// SIMATIC S7-200 project (STEP 7-Micro/WIN), CPU 222 REL 01.22

SYMBOL_TABLE USR1
手动上升I            I0.0     // 用做手动上升，有故障时做故障复位用，常开
手动下降I            I0.1     // 用做手动下降，有故障时做故障复位用，常开
上限位I             I0.2     // 常闭
下限位I             I0.3     // 常闭
启动I              I0.4     // 常开
超时输入I            I0.5     // 来自转子短接接触器，常闭
超温输入I            I0.6     // 常开
上升输出Q            Q0.0     // 上升接触器
下降输出Q            Q0.1     // 下降接触器
允许起动Q            Q0.2     // 给高压柜的允许起动信号
超时跳闸Q            Q0.3     // 包括液体柜电极下降超时及短接接触器超时
转子短接Q            Q0.4
超温报警Q            Q0.5
上升中继M            M1.0     // 调用手动子程序过度用
下降中继M            M1.1     // 调用手动子程序过度用
起动中继M            M1.2     // 调用自动子程序过度用
定时搅拌M            M1.3     // 防止粉沉淀
END_SYMBOL_TABLE

ORGANIZATION_BLOCK 主:OB1
TITLE= 
// 程序注释
// 按 F1 获得帮助及举例程序
//  
BEGIN
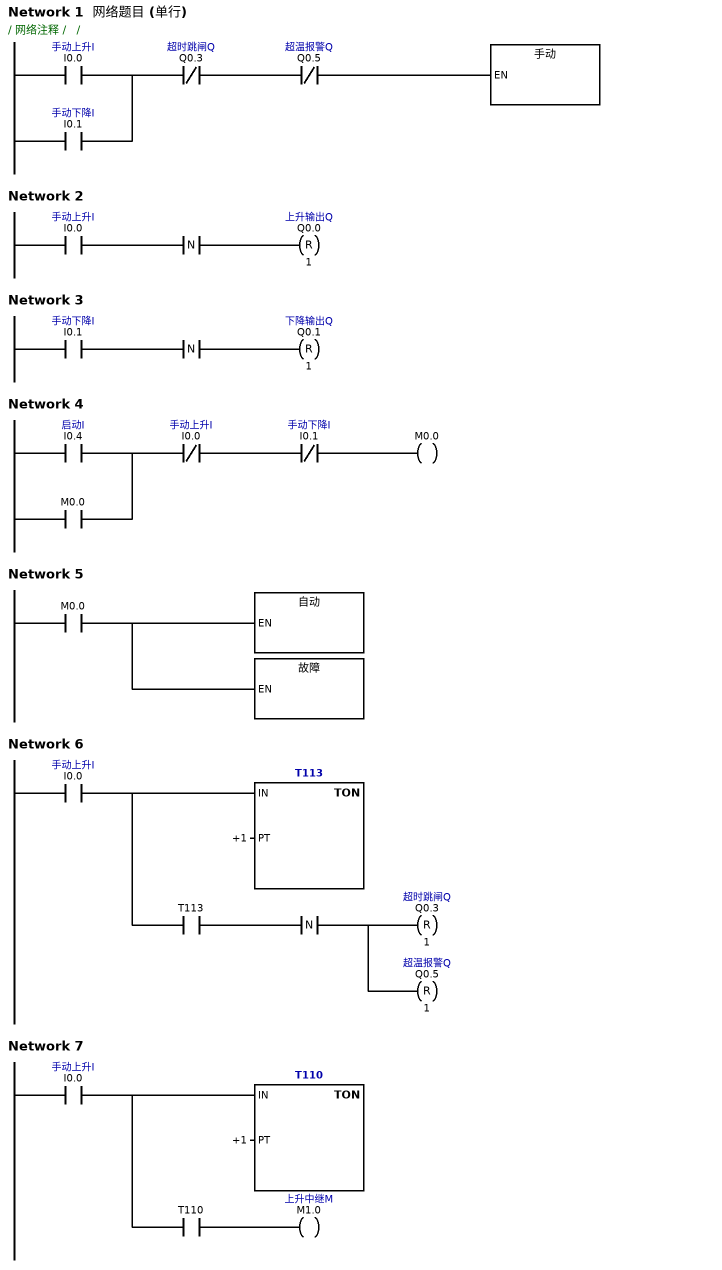
Network 1 // 网络题目 (单行)
//  
// 网络注释
//  
// 
// (network saved uncompiled; LAD cells follow)
// row 0: c0 -| |- 手动上升I:I0.0 v  c1 -|/|- 超时跳闸Q:Q0.3  c2 -|/|- 超温报警Q:Q0.5  c3 --  c4 [手动 EN:=power@row0]
// row 1: c0 -| |- 手动下降I:I0.1 ^
Network 2
// (network saved uncompiled; LAD cells follow)
// row 0: c0 -| |- 手动上升I:I0.0  c1 -|N|-  c2 -(R) 上升输出Q:Q0.0, 1
Network 3
// (network saved uncompiled; LAD cells follow)
// row 0: c0 -| |- 手动下降I:I0.1  c1 -|N|-  c2 -(R) 下降输出Q:Q0.1, 1
Network 4
// (network saved uncompiled; LAD cells follow)
// row 0: c0 -| |- 启动I:I0.4 v  c1 -|/|- 手动上升I:I0.0  c2 -|/|- 手动下降I:I0.1  c3 -( ) M0.0
// row 1: c0 -| |- M0.0 ^
Network 5
// (network saved uncompiled; LAD cells follow)
// row 0: c0 -| |- M0.0 v  c1 --  c2 [自动 EN:=power@row0]
// row 1: c0 ^  c1 --  c2 [故障 EN:=power@row1]
Network 6
// (network saved uncompiled; LAD cells follow)
// row 0: c0 -| |- 手动上升I:I0.0 v  c1 --  c2 [TON T113 IN:=power@row0, PT:=+1]
// row 1: c0 ^v  c2 [box]
// row 2: c0 ^  c1 -| |- T113  c2 -|N|-  v  c3 -(R) 超时跳闸Q:Q0.3, 1
// row 3: c2 ^  c3 -(R) 超温报警Q:Q0.5, 1
Network 7
// (network saved uncompiled; LAD cells follow)
// row 0: c0 -| |- 手动上升I:I0.0 v  c1 --  c2 [TON T110 IN:=power@row0, PT:=+1]
// row 1: c0 ^v  c2 [box]
// row 2: c0 ^  c1 -| |- T110  c2 -( ) 上升中继M:M1.0
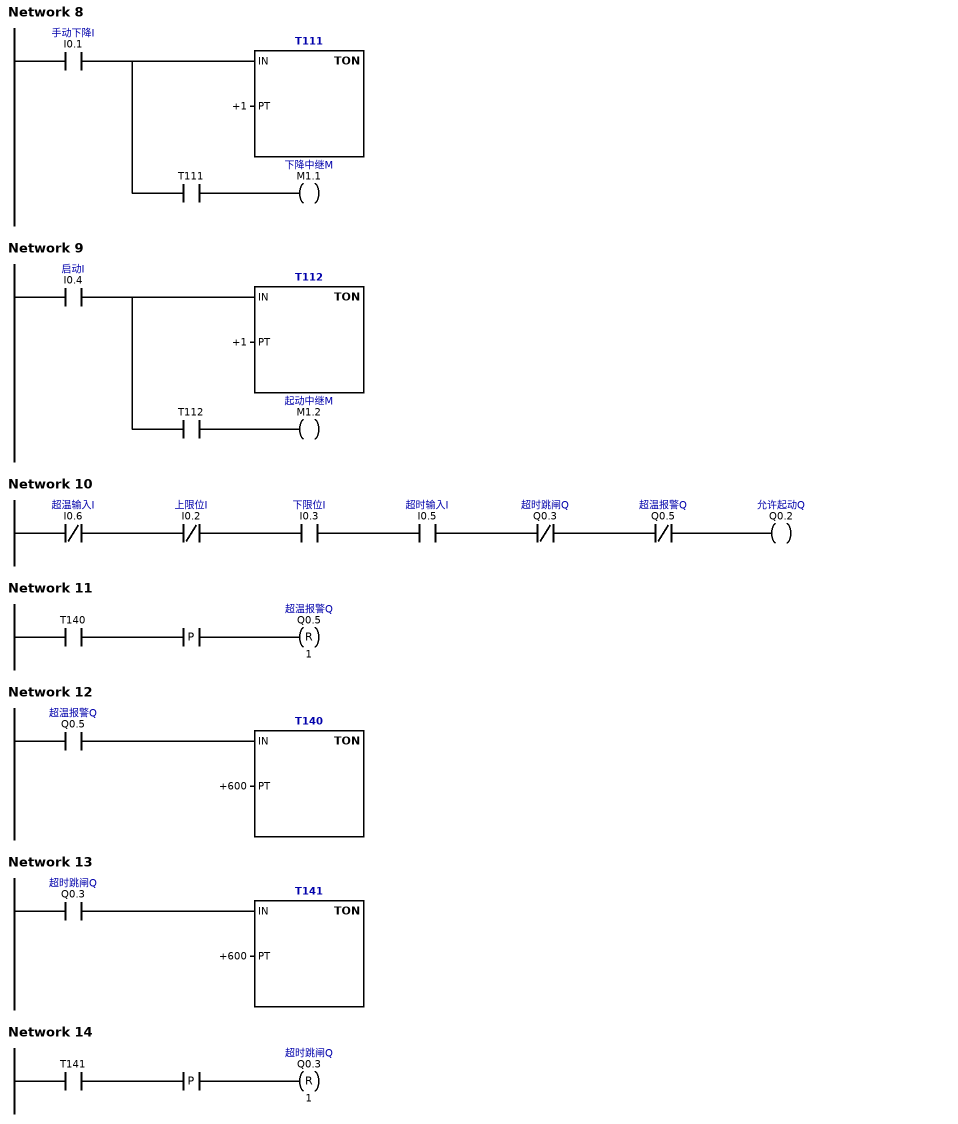
Network 8
// (network saved uncompiled; LAD cells follow)
// row 0: c0 -| |- 手动下降I:I0.1 v  c1 --  c2 [TON T111 IN:=power@row0, PT:=+1]
// row 1: c0 ^v  c2 [box]
// row 2: c0 ^  c1 -| |- T111  c2 -( ) 下降中继M:M1.1
Network 9
// (network saved uncompiled; LAD cells follow)
// row 0: c0 -| |- 启动I:I0.4 v  c1 --  c2 [TON T112 IN:=power@row0, PT:=+1]
// row 1: c0 ^v  c2 [box]
// row 2: c0 ^  c1 -| |- T112  c2 -( ) 起动中继M:M1.2
Network 10
// (network saved uncompiled; LAD cells follow)
// row 0: c0 -|/|- 超温输入I:I0.6  c1 -|/|- 上限位I:I0.2  c2 -| |- 下限位I:I0.3  c3 -| |- 超时输入I:I0.5  c4 -|/|- 超时跳闸Q:Q0.3  c5 -|/|- 超温报警Q:Q0.5  c6 -( ) 允许起动Q:Q0.2
Network 11
// (network saved uncompiled; LAD cells follow)
// row 0: c0 -| |- T140  c1 -|P|-  c2 -(R) 超温报警Q:Q0.5, 1
Network 12
// (network saved uncompiled; LAD cells follow)
// row 0: c0 -| |- 超温报警Q:Q0.5  c1 --  c2 [TON T140 IN:=power@row0, PT:=+600]
// row 1: c2 [box]
Network 13
// (network saved uncompiled; LAD cells follow)
// row 0: c0 -| |- 超时跳闸Q:Q0.3  c1 --  c2 [TON T141 IN:=power@row0, PT:=+600]
// row 1: c2 [box]
Network 14
// (network saved uncompiled; LAD cells follow)
// row 0: c0 -| |- T141  c1 -|P|-  c2 -(R) 超时跳闸Q:Q0.3, 1
END_ORGANIZATION_BLOCK

SUBROUTINE_BLOCK ê??ˉ:SBR0
TITLE= 
// 子程序注释
// 按 F1 获得帮助及举例程序
//  
BEGIN
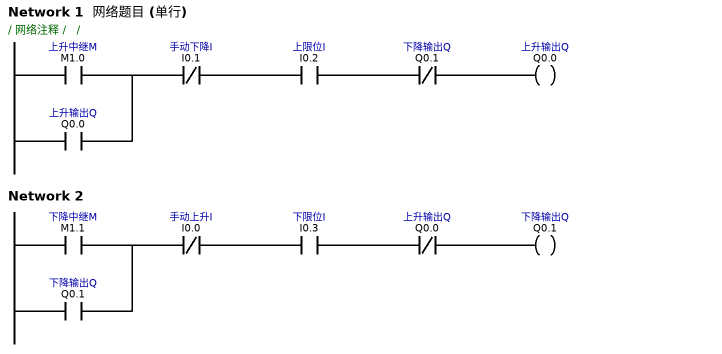
Network 1 // 网络题目 (单行)
//  
// 网络注释
//  
// 
// (network saved uncompiled; LAD cells follow)
// row 0: c0 -| |- 上升中继M:M1.0 v  c1 -|/|- 手动下降I:I0.1  c2 -| |- 上限位I:I0.2  c3 -|/|- 下降输出Q:Q0.1  c4 -( ) 上升输出Q:Q0.0
// row 1: c0 -| |- 上升输出Q:Q0.0 ^
Network 2
// (network saved uncompiled; LAD cells follow)
// row 0: c0 -| |- 下降中继M:M1.1 v  c1 -|/|- 手动上升I:I0.0  c2 -| |- 下限位I:I0.3  c3 -|/|- 上升输出Q:Q0.0  c4 -( ) 下降输出Q:Q0.1
// row 1: c0 -| |- 下降输出Q:Q0.1 ^
END_SUBROUTINE_BLOCK

SUBROUTINE_BLOCK ×??ˉ:SBR1
TITLE=
BEGIN
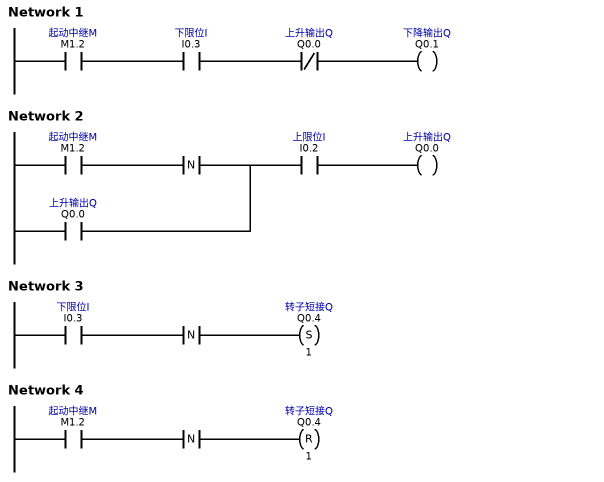
Network 1
// (network saved uncompiled; LAD cells follow)
// row 0: c0 -| |- 起动中继M:M1.2  c1 -| |- 下限位I:I0.3  c2 -|/|- 上升输出Q:Q0.0  c3 -( ) 下降输出Q:Q0.1
Network 2
// (network saved uncompiled; LAD cells follow)
// row 0: c0 -| |- 起动中继M:M1.2  c1 -|N|-  v  c2 -| |- 上限位I:I0.2  c3 -( ) 上升输出Q:Q0.0
// row 1: c0 -| |- 上升输出Q:Q0.0  c1 -- ^
Network 3
// (network saved uncompiled; LAD cells follow)
// row 0: c0 -| |- 下限位I:I0.3  c1 -|N|-  c2 -(S) 转子短接Q:Q0.4, 1
Network 4
// (network saved uncompiled; LAD cells follow)
// row 0: c0 -| |- 起动中继M:M1.2  c1 -|N|-  c2 -(R) 转子短接Q:Q0.4, 1
END_SUBROUTINE_BLOCK

SUBROUTINE_BLOCK 1ê??:SBR2
TITLE=
BEGIN
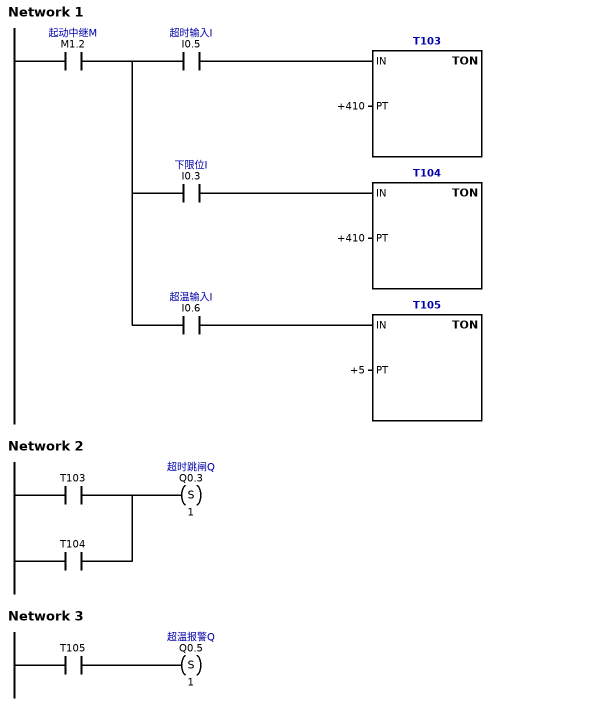
Network 1
// (network saved uncompiled; LAD cells follow)
// row 0: c0 -| |- 起动中继M:M1.2 v  c1 -| |- 超时输入I:I0.5  c2 --  c3 [TON T103 IN:=power@row0, PT:=+410]
// row 1: c0 ^v  c3 [box]
// row 2: c0 ^v  c1 -| |- 下限位I:I0.3  c2 --  c3 [TON T104 IN:=power@row2, PT:=+410]
// row 3: c0 ^v  c3 [box]
// row 4: c0 ^  c1 -| |- 超温输入I:I0.6  c2 --  c3 [TON T105 IN:=power@row4, PT:=+5]
// row 5: c3 [box]
Network 2
// (network saved uncompiled; LAD cells follow)
// row 0: c0 -| |- T103 v  c1 -(S) 超时跳闸Q:Q0.3, 1
// row 1: c0 -| |- T104 ^
Network 3
// (network saved uncompiled; LAD cells follow)
// row 0: c0 -| |- T105  c1 -(S) 超温报警Q:Q0.5, 1
END_SUBROUTINE_BLOCK
